// TwinCAT 3 PLC project PlcSample_IpcDiag
// ProgramVersion: 3.1.4020.4
// libraries:
//   Tc2_Standard, * (Beckhoff Automation GmbH)
//   Tc2_System, * (Beckhoff Automation GmbH)
//   Tc3_IPCDiag, * (Beckhoff Automation GmbH)
//   Tc3_Module, * (Beckhoff Automation GmbH)
// project tree:
//   DUTs/ E_State.TcDUT
//   / PlcTask.TcTTO
//   POUs/ IpcDiagnostics.TcPOU, MAIN.TcPOU, IpcDiagnostics_2.TcPOU
// real-time tasks:
//   TASK PlcTask: cycle T#10ms, priority 20, ADS port 350

CONFIGURATION PlcSample_IpcDiag
    RESOURCE PLC ON TwinCAT3
        TASK PlcTask(INTERVAL := T#10ms, PRIORITY := 20);
        PROGRAM MAIN WITH PlcTask : MAIN;
    END_RESOURCE
END_CONFIGURATION

// ---- DUTs/E_State.TcDUT
{attribute 'qualified_only'}
TYPE E_State :
(
	Init := 0,
	ReadOnce,
	ReadPeriodically,
	Error,
	
	Idle,
	ReadOnce_CpuUsage,
	ReadOnce_CpuTemperature,
	ReadOnce_SrnMainboard,
	ReadOnce_SrnIPC,
	Write_DHCP,
	Write_IPAddr
	
);
END_TYPE

// ---- POUs/MAIN.TcPOU
PROGRAM MAIN
VAR
	i : INT;
END_VAR

i := i + 1;

IpcDiagnostics();		// first way to implement the IPC diagnostics

IpcDiagnostics_2();		// second way to implement the IPC diagnostics

END_PROGRAM

// ---- POUs/IpcDiagnostics.TcPOU
PROGRAM IpcDiagnostics
VAR CONSTANT
	cNetId			: T_AmsNetID := '';				// local
	cNbrParameters	: UDINT := 8;					// number of parameters to read 
END_VAR
VAR
	bStart			: BOOL := TRUE;       			// flag to trigger (re)start of statemachine
	eState			: E_State := E_State.Init;
	hrGetValue		: HRESULT;	

	sDeviceName		: STRING(39);
	nCpuFreq		: UDINT;
	nTcBuild		: UINT;
	aNetworkNames	: ARRAY[1..3] OF STRING(79);	// array in order to receive info of up to three network ports (NICs)
	aIpAddr			: ARRAY[1..3] OF STRING(39);	// array in order to receive info of up to three network ports (NICs)
	aDHCP			: ARRAY[1..3] OF BOOL;			// array in order to receive info of up to three network ports (NICs)
	sMdpVersion		: STRING;
	nBootCnt		: UDINT;
	
	nCpuTemperature	: INT;							// [°C]; should be read periodically
	

	fbDiagRegister	: FB_IPCDiag_Register := (sNetId:=cNetId);
	fbDiagRead		: FB_IPCDiag_ReadParameter := (sNetId:=cNetId);
	nKeyIdx			: USINT := 1;
	aParameterKeys	: ARRAY[1..cNbrParameters] OF E_IPCDiag_ParameterKey := [	E_IPCDiag_ParameterKey.IPCDeviceName,
																				E_IPCDiag_ParameterKey.CPU_Frequency,
																				E_IPCDiag_ParameterKey.TC_VersionBuild,
																				E_IPCDiag_ParameterKey.NIC_Name,
																				E_IPCDiag_ParameterKey.NIC_IPv4Address,
																				E_IPCDiag_ParameterKey.NIC_DHCP,
																				E_IPCDiag_ParameterKey.Software_MDPVersion,
																				E_IPCDiag_ParameterKey.MB_BootCnt ];
	fbDiagReadPeriodic : FB_IPCDiag_ReadParameterPeriodic := (eParameterKey:=E_IPCDiag_ParameterKey.CPU_Temp, tPeriod:= T#10S, sNetId:=cNetId);
END_VAR


CASE eState OF
E_State.Init:
	IF NOT fbDiagRegister.bBusy THEN
		fbDiagRegister(bExecute:=TRUE); // need to be executed once
	ELSE
		fbDiagRegister(bExecute:=FALSE);
	END_IF
	IF NOT fbDiagRegister.bBusy THEN
		IF fbDiagRegister.bError THEN
			eState := E_State.Error;
		ELSE
			eState := E_State.Idle;
		END_IF
	END_IF

E_State.Idle:
    IF bStart THEN
        bStart := FALSE;
        eState := E_State.ReadOnce;
    END_IF

E_State.ReadOnce: // reads every parameter once
	IF NOT fbDiagRead.bBusy THEN
		fbDiagRead(bExecute:= TRUE, eParameterKey:=aParameterKeys[nKeyIdx], fbRegister:=fbDiagRegister);	
	ELSE
		fbDiagRead(bExecute:= FALSE, fbRegister:=fbDiagRegister);
	END_IF
	IF NOT fbDiagRead.bBusy THEN
		IF fbDiagRead.bError THEN
			eState := E_State.Error;
		ELSE // get value
			IF aParameterKeys[nKeyIdx] = E_IPCDiag_ParameterKey.IPCDeviceName THEN
				hrGetValue := fbDiagRead.GetParameter(pBuffer:=ADR(sDeviceName), nBufferSize:=SIZEOF(sDeviceName));
				
			ELSIF aParameterKeys[nKeyIdx] = E_IPCDiag_ParameterKey.CPU_Frequency THEN
				hrGetValue := fbDiagRead.GetParameter(pBuffer:=ADR(nCpuFreq), nBufferSize:=SIZEOF(nCpuFreq));
				
			ELSIF aParameterKeys[nKeyIdx] = E_IPCDiag_ParameterKey.TC_VersionBuild THEN
				hrGetValue := fbDiagRead.GetParameter(pBuffer:=ADR(nTcBuild), nBufferSize:=SIZEOF(nTcBuild));
				
			ELSIF aParameterKeys[nKeyIdx] = E_IPCDiag_ParameterKey.NIC_Name THEN
				// get values (one by one)
				hrGetValue := fbDiagRead.GetParameterByIdx(pBuffer:=ADR(aNetworkNames[1]), nBufferSize:=SIZEOF(aNetworkNames[1]), 1);
				IF SUCCEEDED(hrGetValue) THEN
					hrGetValue := fbDiagRead.GetParameterByIdx(pBuffer:=ADR(aNetworkNames[2]), nBufferSize:=SIZEOF(aNetworkNames[2]), 2);
				END_IF
				IF SUCCEEDED(hrGetValue) THEN
					hrGetValue := fbDiagRead.GetParameterByIdx(pBuffer:=ADR(aNetworkNames[3]), nBufferSize:=SIZEOF(aNetworkNames[3]), 3);
				END_IF
				
			ELSIF aParameterKeys[nKeyIdx] = E_IPCDiag_ParameterKey.NIC_IPv4Address THEN
				// get values (all together)
				hrGetValue := fbDiagRead.GetParameterStrings(pBuffer:=ADR(aIpAddr), nBufferSize:=SIZEOF(aIpAddr), nStrings:=3);
				
			ELSIF aParameterKeys[nKeyIdx] = E_IPCDiag_ParameterKey.NIC_DHCP THEN
				// get values (all together)
				hrGetValue := fbDiagRead.GetParameter(pBuffer:=ADR(aDHCP), nBufferSize:=SIZEOF(aDHCP));
				
			ELSIF aParameterKeys[nKeyIdx] = E_IPCDiag_ParameterKey.Software_MDPVersion THEN
				hrGetValue := fbDiagRead.GetParameter(pBuffer:=ADR(sMdpVersion), nBufferSize:=SIZEOF(sMdpVersion));
			
			ELSIF aParameterKeys[nKeyIdx] = E_IPCDiag_ParameterKey.MB_BootCnt THEN
				hrGetValue := fbDiagRead.GetParameter(pBuffer:=ADR(nBootCnt), nBufferSize:=SIZEOF(nBootCnt));
			
			END_IF
				
			IF SUCCEEDED(hrGetValue) THEN
				IF nKeyIdx = cNbrParameters THEN // all keys successfully read
					nKeyIdx := 1;
					eState := E_State.ReadPeriodically;
				ELSE
					nKeyIdx := nKeyIdx + 1;
				END_IF
			ELSE
				eState := E_State.Error;
			END_IF
		END_IF
	END_IF	

E_State.ReadPeriodically:
	fbDiagReadPeriodic(bEnable:=TRUE, fbRegister:=fbDiagRegister);
	IF fbDiagReadPeriodic.bValid THEN
		fbDiagReadPeriodic.GetParameter(pBuffer:=ADR(nCpuTemperature), nBufferSize:=SIZEOF(nCpuTemperature) );	
	END_IF
	IF fbDiagReadPeriodic.bError THEN
		eState := E_State.Error;
	END_IF	
	
E_State.Error:
	(* implementation of error logging and error handling *)
	(* hint: An error could also occur if a parameter is not supported by chosen hardware or image. 
	E.g. not all IPCs offer a CPU temperature measurement. *)

END_CASE

END_PROGRAM

// ---- POUs/IpcDiagnostics_2.TcPOU
PROGRAM IpcDiagnostics_2
VAR CONSTANT
	cNetId					: T_AmsNetID := '';		// local
END_VAR
VAR
    bStart              	: BOOL := TRUE;       	// flag to trigger (re)start of statemachine
	bSkipSettingIPAddr		: BOOL := TRUE;			// for safety reasons - set FALSE if you want to set the IP address
	eState					: E_State := E_State.Init;
	
    bError              	: BOOL;               	// error flag (indicator: error occured)
    hrErrorCode             : HRESULT;             	// last error code
	hrGetValue				: HRESULT;
	
    nCpuUsage           	: UINT;               	// CPU usage [%]
	nCpuTemperature			: INT;					// CPU temperature [°C]
    sSerialNumberMainboard	: STRING;       		// serial number of mainboard
    sSerialNumberIPC        : STRING;          		// serial number of IPC
	nNicModuleIdx			: USINT := 1;			// select which NIC adapter should be adapted with a new IP address
    bDHCP					: BOOL := FALSE;
	sIPAddr			        : T_IPv4Addr := '174.18.3.154'; // the new ip address 
    aFanSpeed           	: ARRAY[1..2] OF UINT;	// speed of fans - should be read periodically
	
	fbDiagRegister			: FB_IPCDiag_Register := (sNetId:=cNetId);
	fbDiagRead				: FB_IPCDiag_ReadParameter := (sNetId:=cNetId);
	fbDiagReadPeriodic		: FB_IPCDiag_ReadParameterPeriodic := (tPeriod:= T#10S, sNetId:=cNetId);
	fbDiagWrite				: FB_IPCDiag_WriteParameter := (sNetId:=cNetId);
END_VAR

CASE eState OF

E_State.Init:
	IF NOT fbDiagRegister.bBusy THEN
		fbDiagRegister(bExecute:=TRUE);
	ELSE
		fbDiagRegister(bExecute:=FALSE, bError=>bError, hrErrorCode=>hrErrorCode);
	END_IF
	IF NOT fbDiagRegister.bBusy THEN
		IF fbDiagRegister.bError THEN
			eState := E_State.Error;
		ELSE
			eState := E_State.Idle;
		END_IF
	END_IF

E_State.Idle:
    IF bStart THEN
        bStart := FALSE;
        eState := E_State.ReadOnce_CpuUsage;
    END_IF

E_State.ReadOnce_CpuUsage:
	IF NOT fbDiagRead.bBusy THEN
		fbDiagRead(bExecute:= TRUE, eParameterKey:=E_IPCDiag_ParameterKey.CPU_Usage, fbRegister:=fbDiagRegister);	
	ELSE
		fbDiagRead(bExecute:= FALSE, fbRegister:=fbDiagRegister, bError=>bError, hrErrorCode=>hrErrorCode);
	END_IF
	IF NOT fbDiagRead.bBusy THEN
		IF fbDiagRead.bError THEN
			eState := E_State.Error;
		ELSE // get value
			hrGetValue := fbDiagRead.GetParameter(pBuffer:=ADR(nCpuUsage), nBufferSize:=SIZEOF(nCpuUsage));	
			IF FAILED(hrGetValue) THEN
				eState := E_State.Error;
			ELSE
				eState := E_State.ReadOnce_CpuTemperature;
			END_IF
		END_IF
	END_IF	

E_State.ReadOnce_CpuTemperature:
	IF NOT fbDiagRead.bBusy THEN
		fbDiagRead(bExecute:= TRUE, eParameterKey:=E_IPCDiag_ParameterKey.CPU_Temp, fbRegister:=fbDiagRegister);	
	ELSE
		fbDiagRead(bExecute:= FALSE, fbRegister:=fbDiagRegister, bError=>bError, hrErrorCode=>hrErrorCode);
	END_IF
	IF NOT fbDiagRead.bBusy THEN
		IF fbDiagRead.bError THEN
			eState := E_State.Error;
		ELSE // get value
			hrGetValue := fbDiagRead.GetParameter(pBuffer:=ADR(nCpuTemperature), nBufferSize:=SIZEOF(nCpuTemperature));	
			IF FAILED(hrGetValue) THEN
				eState := E_State.Error;
			ELSE
				eState := E_State.ReadOnce_SrnMainboard;
			END_IF
		END_IF
	END_IF

E_State.ReadOnce_SrnMainboard:
	IF NOT fbDiagRead.bBusy THEN
		fbDiagRead(bExecute:= TRUE, eParameterKey:=E_IPCDiag_ParameterKey.MB_SerialNumber, fbRegister:=fbDiagRegister);	
	ELSE
		fbDiagRead(bExecute:= FALSE, fbRegister:=fbDiagRegister, bError=>bError, hrErrorCode=>hrErrorCode);
	END_IF
	IF NOT fbDiagRead.bBusy THEN
		IF fbDiagRead.bError THEN
			eState := E_State.Error;
		ELSE // get value
			hrGetValue := fbDiagRead.GetParameter(pBuffer:=ADR(sSerialNumberMainboard), nBufferSize:=SIZEOF(sSerialNumberMainboard));	
			IF FAILED(hrGetValue) THEN
				eState := E_State.Error;
			ELSE
				eState := E_State.ReadOnce_SrnIPC;
			END_IF
		END_IF
	END_IF

E_State.ReadOnce_SrnIPC:
	IF NOT fbDiagRead.bBusy THEN
		fbDiagRead(bExecute:= TRUE, eParameterKey:=E_IPCDiag_ParameterKey.IPCSerialNumber, fbRegister:=fbDiagRegister);	
	ELSE
		fbDiagRead(bExecute:= FALSE, fbRegister:=fbDiagRegister, bError=>bError, hrErrorCode=>hrErrorCode);
	END_IF
	IF NOT fbDiagRead.bBusy THEN
		IF fbDiagRead.bError THEN
			eState := E_State.Error;
		ELSE // get value
			hrGetValue := fbDiagRead.GetParameter(pBuffer:=ADR(sSerialNumberIPC), nBufferSize:=SIZEOF(sSerialNumberIPC));	
			IF FAILED(hrGetValue) THEN
				eState := E_State.Error;
			ELSE
				IF bSkipSettingIPAddr THEN
					eState := E_State.ReadPeriodically;
				ELSE
					eState := E_State.Write_DHCP;
				END_IF
			END_IF
		END_IF
	END_IF

E_State.Write_DHCP:
	IF NOT fbDiagWrite.bBusy THEN
		fbDiagWrite(bExecute:= TRUE, 
					eParameterKey:=E_IPCDiag_ParameterKey.NIC_DHCP,
					pBuffer:=ADR(bDHCP),
					nBufferSize:=SIZEOF(bDHCP),
					nModuleIdx:=nNicModuleIdx,
					fbRegister:=fbDiagRegister );	
	ELSE
		fbDiagWrite(bExecute:= FALSE, fbRegister:=fbDiagRegister, bError=>bError, hrErrorCode=>hrErrorCode);
	END_IF
	IF NOT fbDiagWrite.bBusy THEN
		IF fbDiagWrite.bError THEN
			eState := E_State.Error;
		ELSE
			eState := E_State.Write_IPAddr;
		END_IF
	END_IF

E_State.Write_IPAddr:
	IF NOT fbDiagWrite.bBusy THEN
		fbDiagWrite(bExecute:= TRUE, 
					eParameterKey:=E_IPCDiag_ParameterKey.NIC_IPv4Address,
					pBuffer:=ADR(sIPAddr),
					nBufferSize:=INT_TO_UDINT(LEN(sIPAddr)+1),
					nModuleIdx:=nNicModuleIdx,
					fbRegister:=fbDiagRegister );	
	ELSE
		fbDiagWrite(bExecute:= FALSE, fbRegister:=fbDiagRegister, bError=>bError, hrErrorCode=>hrErrorCode);
	END_IF
	IF NOT fbDiagWrite.bBusy THEN
		IF fbDiagWrite.bError THEN
			eState := E_State.Error;
		ELSE
			eState := E_State.ReadPeriodically;
		END_IF
	END_IF

E_State.ReadPeriodically:
	fbDiagReadPeriodic(bEnable:=TRUE, eParameterKey:=E_IPCDiag_ParameterKey.Fan_Speed, fbRegister:=fbDiagRegister, bError=>bError, hrErrorCode=>hrErrorCode);
	IF fbDiagReadPeriodic.bValid THEN
		fbDiagReadPeriodic.GetParameter(pBuffer:=ADR(aFanSpeed), nBufferSize:=SIZEOF(aFanSpeed) );	
	END_IF
	IF fbDiagReadPeriodic.bError THEN
		eState := E_State.Error;
	END_IF

E_State.Error:
	(* implementation of error logging and error handling *)
	(* hint: An error could also occur if a parameter is not supported by chosen hardware or image. 
	E.g. not all IPCs offer a CPU temperature measurement. *)
END_CASE

END_PROGRAM
